FUNCTION Convert_USINT_TO_INT : Hresult
VAR_INPUT
	in : USINT;
	out : REFERENCE TO INT;
END_VAR
VAR
	converted : INT;
END_VAR

converted := USINT_TO_INT(in);

IF (INT_TO_USINT(converted) <> in) THEN
	Convert_USINT_TO_INT := INCOMPATIBLE;
	RETURN;
END_IF

out := converted;

END_FUNCTION

(* stored: Version 1.1.0.1, ProductVersion 3.1.4024.12
   POU Convert_USINT_TO_INT: Id {a58865ff-d006-4084-bb33-b378f3695cfc}, SpecialFunc None *)
